{attribute 'GeneratedUsingTerminal: EL6001-0000-0020'}
{attribute addProperty BoxType "EL6001-0000-0020"}
{attribute addProperty Id "InputsAT %I*Inputs_37C8E74C6OutputsAT %Q*Outputs_2CF06B6A6WcStateAT %I*WcState_9091E0EB2InfoDataAT %I*InfoData_94A18F5E2"}
{attribute addProperty CRC "3036469869"}
{attribute addProperty Size "16"}
TYPE EL6001_B4FCDA6D EXTENDS EtcSlaveTerminalBase_947E5A46 :
STRUCT
	{attribute addProperty Name "Inputs"}
	Inputs : Inputs_37C8E74C;
	{attribute addProperty Name "Outputs"}
	Outputs : Outputs_2CF06B6A;
	{attribute addProperty Name "WcState"}
	WcState : WcState_9091E0EB;
	{attribute addProperty Name "InfoData"}
	InfoData : InfoData_94A18F5E;
END_STRUCT
END_TYPE

(* stored: Version 1.2.0.0, ProductVersion 3.1.4024.9
   DUT EL6001_B4FCDA6D: Id {fba01c2e-579d-4c11-9725-31c0013e0af8} *)
